TYPE ST_JogMotorControl :
STRUCT
  bMoveFW   : BOOL := false;
  bMoveBW   : BOOL := false;
END_STRUCT
END_TYPE

(* stored: Version 1.1.0.1, ProductVersion 3.1.4024.12
   DUT ST_JogMotorControl: Id {4133f033-568f-4e26-b326-f74290a7e19f} *)
